SUBAPPLICATION MinusMinus (* Subapplication Type *)
  (* Standard: 61499-2 *)
  (* Version 1.0, 2023-02-17, Franz *)
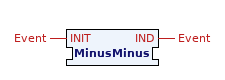
  EVENT_INPUT
    INIT;
  END_EVENT
  EVENT_OUTPUT
    IND;
  END_EVENT
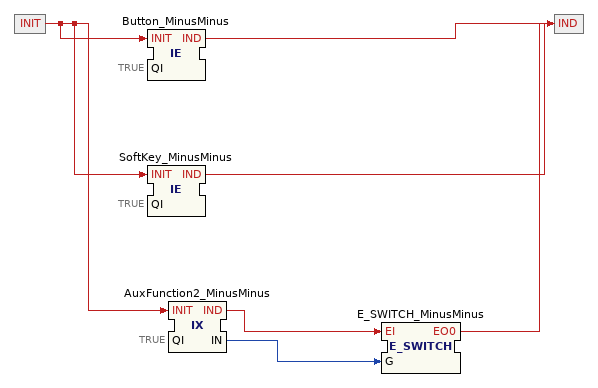
  FBS
    Button_MinusMinus : IE(QI := TRUE);
    SoftKey_MinusMinus : IE(QI := TRUE);
    AuxFunction2_MinusMinus : IX(QI := TRUE);
    E_SWITCH_MinusMinus : E_SWITCH;
  END_FBS
  EVENT_CONNECTIONS
    INIT TO Button_MinusMinus.INIT;
    Button_MinusMinus.IND TO IND;
    INIT TO SoftKey_MinusMinus.INIT;
    SoftKey_MinusMinus.IND TO IND;
    INIT TO AuxFunction2_MinusMinus.INIT;
    AuxFunction2_MinusMinus.IND TO E_SWITCH_MinusMinus.EI;
    E_SWITCH_MinusMinus.EO0 TO IND;
  END_CONNECTIONS
  DATA_CONNECTIONS
    AuxFunction2_MinusMinus.IN TO E_SWITCH_MinusMinus.G;
  END_CONNECTIONS
END_SUBAPPLICATION
